(* IEC 61131-3 sources: UAH_ENG/CPE 459/OpenPLC/Lab_1_First_SCADA, 2 files *)

(* ---- assignment1.st ---- *)
PROGRAM Lab1
  VAR
    PB1 AT %IX100.0 : BOOL;
    PB2 AT %IX100.1 : BOOL;
    LED AT %QX100.0 : BOOL;
  END_VAR

  LED := NOT(PB2) AND (LED OR PB1);
END_PROGRAM

CONFIGURATION Config0

  RESOURCE Res0 ON PLC
    TASK task0(INTERVAL := T#20ms,PRIORITY := 0);
    PROGRAM instance0 WITH task0 : Lab1;
  END_RESOURCE
END_CONFIGURATION

(* ---- hw1.st ---- *)
PROGRAM Lab1
  VAR
    PB1 AT %IX100.0 : BOOL;
    PB2 AT %IX100.1 : BOOL;
    LED AT %QX100.0 : BOOL;
  END_VAR

  LED := NOT(PB2) AND (LED OR PB1);
END_PROGRAM

CONFIGURATION Config0

  RESOURCE Res0 ON PLC
    TASK task0(INTERVAL := T#20ms,PRIORITY := 0);
    PROGRAM instance0 WITH task0 : Lab1;
  END_RESOURCE
END_CONFIGURATION
